//{attribute 'qualified_only'}
VAR_GLOBAL
    (*ETHERCAT BRRIDGE COM STATUS*)
    //0: Other side is in OP state, >0: Error
    {attribute 'TcLinkTo' := 'TIIB[R19_DRL_02_E3_EL6695]^SYNC Inputs^TxPDO state
    '}
    xEcatBridge_TxPDO_state AT %I* :BOOL;

    //0: External device connectd, 1: External device not connected

    {attribute := 'TIIB[R19_DRL_02_E3_EL6695]^SYNC Inputs^External device not connected
    '}
    xEcatBridge_External_device_not_connected AT %I* : BOOL;

    //0 = Data valid, 1 = Data invalid
    {attribute 'TcLinkTo' := 'TIIB[R19_DRL_02_E3_EL6695]^WcState^WcState
    '}
    xEcatBridge_WcState AT %I* : BOOL;

    {attribute 'TcLinkTo' := 'TIIB[R19_DRL_02_E3_EL6695]^IO Inputs^DREAM_VRC_DP1_OPEN_LS'}
    bDREAM_VRC_DP1_OPEN_LS  AT %I* : BOOL;

    {attribute  'TcLinkTo' := 'TIIB[R19_DRL_02_E3_EL6695]^IO Outputs^DREAM_GNZ_Y_OUT'}
    xDREAM_GNZ_Y_OUT AT %Q*: BOOL;

    {attribute  'TcLinkTo' := 'TIIB[R19_DRL_02_E3_EL6695]^IO Outputs^DREAM_GNZ_Y_Ext_OUT'}
    xDREAM_GNZ_Y_Ext_OUT AT %Q*: BOOL;
END_VAR

(* stored: Version 1.1.0.1
   GVL GVL_PLC_Interfaces: Id {b4d32037-6176-4da1-a9af-c4baba1b3a23} *)
